// TIA Portal project "FactoryIO_Template_S7-1200_V15_V17" (V17)
// Vorlageprojekt für das Buch mit Zielsystem S7-1200

(* hardware
DEVICE "S7-1200-Station_1"  S7-1200 Station
   slot 0: "Baugruppenträger_0"  Rack  V1.0
   slot 1: "PLC_1"  CPU 1211C DC/DC/DC  6ES7 211-1AE40-0XB0  V4.1
*)

// ===== PLC "PLC_1"  CPU 1211C DC/DC/DC =====

VAR_GLOBAL   // PLC tag table "Standard-Variablentabelle"
   "Tag_1" AT %A0.0 : Bool;
   "Tag_2" AT %E0.0 : Bool;
   "Tag_3" AT %E0.1 : Bool;
   "Tag_4" AT %I0.4 : Bool;
   "Tag_5" AT %Q1.3 : Bool;
   "Tag_6" AT %Q1.4 : Bool;
   "Tag_7" AT %M0.0 : Bool;
   "Tag_8" AT %I0.3 : Bool;
   "Tag_9" AT %ID30 : DWord;
   "Tag_10" AT %Q0.3 : Bool;
   "Tag_11" AT %M0.1 : Bool;
   "Tag_12" AT %MW0 : Word;
   "Tag_13" AT %Q0.2 : Bool;
   "Tag_14" AT %Q1.5 : Bool;
   "Tag_15" AT %Q0.5 : Bool;
   "Tag_16" AT %Q0.4 : Bool;
   "Tag_17" AT %Q0.6 : Bool;
   "Tag_18" AT %Q0.7 : Bool;
   "Tag_19" AT %Q1.0 : Bool;
   "Tag_20" AT %QD34 : DWord;
END_VAR

// folder: System blocks/Program resources

DATA_BLOCK "IEC_Timer_0_DB"   // DB1
{ S7_Optimized_Access := 'TRUE' }
AUTHOR : Simatic
FAMILY : IEC
NAME : IEC_TMR
VERSION : 1.0
// stored: InstanceOfName IEC_TIMER
"IEC_TIMER"
BEGIN
END_DATA_BLOCK

DATA_BLOCK "IEC_Timer_0_DB_1"   // DB2
{ S7_Optimized_Access := 'TRUE' }
AUTHOR : Simatic
FAMILY : IEC
NAME : IEC_TMR
VERSION : 1.0
// stored: InstanceOfName IEC_TIMER
"IEC_TIMER"
BEGIN
END_DATA_BLOCK

DATA_BLOCK "IEC_Timer_0_DB_2"   // DB3
{ S7_Optimized_Access := 'TRUE' }
AUTHOR : Simatic
FAMILY : IEC
NAME : IEC_TMR
VERSION : 1.0
// stored: InstanceOfName IEC_TIMER
"IEC_TIMER"
BEGIN
END_DATA_BLOCK

// folder: (top level)

FUNCTION "MHJ-PLC-Lab-Function-S71200" : Void   // FC9000, SCL
{ S7_Optimized_Access := 'TRUE' }
VERSION : 0.1
   VAR_TEMP
      rdTimeReturn : Int;
      outputTime : DTL;
      SyncVal : Byte;
      forVal : Int;
      forVal_2 : Int;
      Value : Byte;
   END_VAR
   VAR CONSTANT
      CompVal : Byte := 16#34;
      Value_01 : Byte := 16#11;
      Value_01_DW : DWord := 16#A165_D992;
      Value_02_DW : DWord := 16#58BE_4401;
   END_VAR
BEGIN

   #Value:=PEEK(area := 16#82,
        dbNumber := 0,
        byteOffset := 511);
   #Value := #Value + 1;

   POKE(area := 16#82,
        dbNumber := 0,
        byteOffset := 511,
        value := #Value);

   POKE(area:=16#81,
        dbNumber:=0,
        byteOffset:=1016,
        value:=#Value_01_DW);
   POKE(area := 16#81,
        dbNumber := 0,
        byteOffset := 1020,
        value := #Value_02_DW);

   POKE(area := 16#81,
        dbNumber := 0,
        byteOffset := 511,
        value := B#16#00);

   FOR #forVal := 0 TO 120 DO
       FOR #forVal_2:=0 TO 10 DO
           #rdTimeReturn:=RD_SYS_T(#outputTime);
           #rdTimeReturn := WR_SYS_T(#outputTime);
           #rdTimeReturn := RD_SYS_T(#outputTime);
           #rdTimeReturn := WR_SYS_T(#outputTime);
       END_FOR;
       #SyncVal:= PEEK(area := 16#81,
                      dbNumber := 0,
                      byteOffset := 511);
       IF #SyncVal = #CompVal THEN
          GOTO M_1;
       END_IF;
   END_FOR;
   RETURN;

   M_1:
   POKE(area := 16#81,
        dbNumber := 0,
        byteOffset := 511,
        value := B#16#0);
END_FUNCTION

ORGANIZATION_BLOCK "Main"   // OB1, LAD, ProgramCycle
TITLE = "Main Program Sweep (Cycle)"
{ S7_Optimized_Access := 'TRUE' }
VERSION : 0.1
   VAR_INPUT
      Initial_Call : Bool;   // Initial call of this OB
      Remanence : Bool;   // =True, if remanent data are available
   END_VAR
   VAR_TEMP
      tacc : Time;
      tacc1 : Time;
      tacc2 : Time;
   END_VAR
BEGIN

REGION Network 1: Konnektierungsbaustein für PLC-Lab
   // Im Netzwerk 1 wird der Konnektierungsbaustein für PLC-Lab aufgerufen.
   // Dieser Aufruf darf nicht entfernt werden!
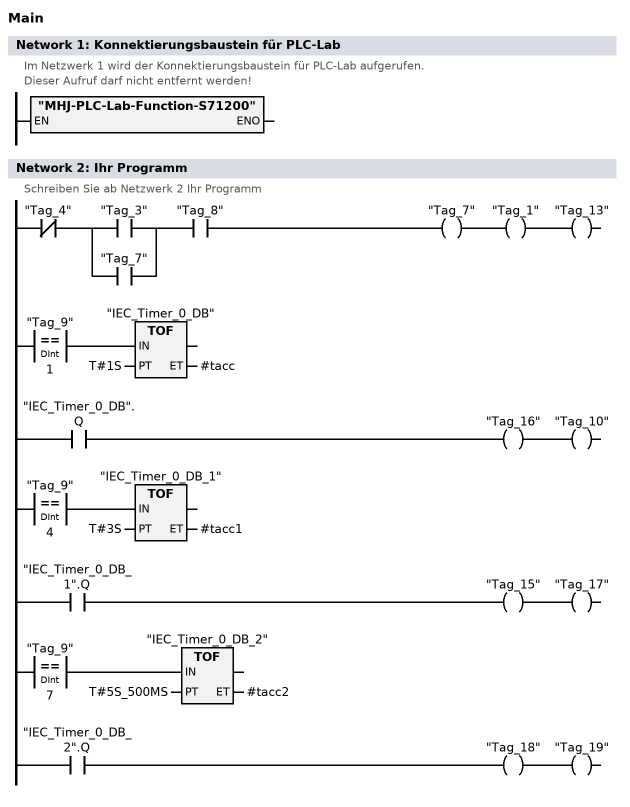
   RUNG wire#powerrail
      "MHJ-PLC-Lab-Function-S71200"()
   END_RUNG
   // the same network as SCL:
   "MHJ-PLC-Lab-Function-S71200"();
END_REGION

REGION Network 2: Ihr Programm
   // Schreiben Sie ab Netzwerk 2 Ihr Programm
   "Tag_7" := NOT "Tag_4" AND ("Tag_3" OR "Tag_7") AND "Tag_8";
   "Tag_1" := "Tag_7";
   "Tag_13" := "Tag_7";
   "IEC_Timer_0_DB".TOF(IN := "Tag_9" = 1, PT := T#1S, ET => #tacc);
   "Tag_16" := "IEC_Timer_0_DB".Q;
   "Tag_10" := "IEC_Timer_0_DB".Q;
   "IEC_Timer_0_DB_1".TOF(IN := "Tag_9" = 4, PT := T#3S, ET => #tacc1);
   "Tag_15" := "IEC_Timer_0_DB_1".Q;
   "Tag_17" := "IEC_Timer_0_DB_1".Q;
   "IEC_Timer_0_DB_2".TOF(IN := "Tag_9" = 7, PT := T#5S_500MS, ET => #tacc2);
   "Tag_18" := "IEC_Timer_0_DB_2".Q;
   "Tag_19" := "IEC_Timer_0_DB_2".Q;
END_REGION
END_ORGANIZATION_BLOCK